// TIA Portal V18 export
DATA_BLOCK "AHUProxyCH"   // DB59021
{ S7_Optimized_Access := 'FALSE' }
VERSION : 0.1
// stored: AutoNumber false, DBAccessibleFromOPCUA true, IsOnlyStoredInLoadMemory false, IsWriteProtectedInAS false
   VAR
      Vars { S7_SetPoint := 'True'} : "UDT_AnalogProxyCH_Vars";
   END_VAR
BEGIN
END_DATA_BLOCK
